METHOD VisitComponent
VAR_INPUT
	Component : Core.I_Component;
END_VAR
_OK := TRUE;
IF __QUERYINTERFACE(Component, SafetyComponent) THEN
	IF NOT SafetyComponent.OK THEN
		ErrorComponent := Component;
		_OK			   := FALSE;
	END_IF
END_IF
END_METHOD

END_FUNCTION_BLOCK

// Components/Safety/Visitor/SetSafetySimulationVisitor
FUNCTION_BLOCK SetSafetySimulationVisitor IMPLEMENTS I_ComponentVisitor
VAR
	SafetyComponent : I_SafetyBase;
	InfoData		: ST_SafetyStateDiag;
	_Simulated		: BOOL;
END_VAR

PROPERTY Diag : UINT
SET
InfoData.Diag := Diag;
END_SET
END_PROPERTY

PROPERTY Simulated : BOOL
GET
Simulated := _Simulated;
END_GET
SET
_Simulated := Simulated;
END_SET
END_PROPERTY

PROPERTY State : USINT
SET
InfoData.State := State;
END_SET
END_PROPERTY

METHOD VisitComponent
VAR_INPUT
	Component : Core.I_Component;
END_VAR
IF __QUERYINTERFACE(Component, SafetyComponent) THEN
	SafetyComponent.Simulated := _Simulated;
	SafetyComponent.SimulateSafetyDiag(InfoData.Diag);
	SafetyComponent.SimulateSafetyState(InfoData.State);
END_IF
END_METHOD

END_FUNCTION_BLOCK

// Components/Safety/SafetyAndOrFB
FUNCTION_BLOCK SafetyAndOrFB EXTENDS SafetyBase
VAR
END_VAR

METHOD CyclicLogic
VAR_INST
	LinkError : BOOL;
END_VAR
SUPER^.CyclicLogic();
_OK := SUPER^.InfoData.State = E_SafetyOrAnd_State.Run;
END_METHOD

END_FUNCTION_BLOCK

// Components/Safety/SafetyBase
FUNCTION_BLOCK SafetyBase EXTENDS CyclicComponent IMPLEMENTS I_SafetyBase
VAR
	InfoData AT %I* : ST_SafetyStateDiag;
	{attribute 'hide'}
	_Simulated : BOOL;
	{attribute 'hide'}
	_OK : BOOL;
	{attribute 'hide'}
	_Error : BOOL;
	{attribute 'hide'}
	_Busy : BOOL;
	{attribute 'hide'}
	_ErrorId	   : UDINT;
	_ResetFunction : I_SafetyReset;
END_VAR

METHOD CyclicLogic
VAR_INST
	LinkError : BOOL;
END_VAR
IF NOT LinkError AND NOT Simulated AND (F_GetMappingStatus(ADR(InfoData), SIZEOF(InfoData)) = EplcMappingStatus.MS_Unmapped) THEN
	LinkError := TRUE;
	Trace.LogMessage(Name, 'Not mapped to Safety, no diagnostics available!');
END_IF

IF _ResetFunction <> 0 THEN
	_ResetFunction.CyclicLogic();
END_IF
END_METHOD

{attribute 'monitoring' := 'call'}
PROPERTY OK : BOOL
GET
OK := _OK;
END_GET
END_PROPERTY

METHOD Reset
IF _ResetFunction <> 0 THEN
	_ResetFunction.Execute();
END_IF
END_METHOD

PROPERTY ResetFunction : I_SafetyReset
SET
_ResetFunction := ResetFunction;
END_SET
END_PROPERTY

{attribute 'monitoring' := 'call'}
PROPERTY Simulated : BOOL
GET
Simulated := _Simulated;
END_GET
SET
_Simulated := Simulated;
END_SET
END_PROPERTY

METHOD SimulateSafetyDiag
VAR_INPUT
	SimulationValueDiag : UINT;
END_VAR
Infodata.Diag := SimulationValueDiag;
END_METHOD

METHOD SimulateSafetyState
VAR_INPUT
	SimulationValueState : USINT;
END_VAR
Infodata.State := SimulationValueState;
END_METHOD

{attribute 'monitoring' := 'call'}
PROPERTY Busy : BOOL
GET
Busy := _Busy;
END_GET
END_PROPERTY

{attribute 'monitoring' := 'call'}
PROPERTY Error : BOOL
GET
Error := _Error;
END_GET
END_PROPERTY

{attribute 'monitoring' := 'call'}
PROPERTY ErrorId : UDINT
GET
ErrorId := _ErrorId;
END_GET
END_PROPERTY

END_FUNCTION_BLOCK

// Components/Safety/SafetyConnectionFB_TcEvents
FUNCTION_BLOCK SafetyConnectionFB_TcEvents EXTENDS SafetyBase IMPLEMENTS I_EventReactionTcEvents
VAR
	Events : TcEventClass('FSoE Connection Events');
END_VAR

METHOD CyclicLogic
VAR_INST
	DiagWord	: WORD;
	BitMaskDiag : WORD := 16#000F;
END_VAR
SUPER^.CyclicLogic();
_OK	   := SUPER^.InfoData.State = E_SafetyConnection_State.Data;
_Error := GetHighestActiveEventReaction() >= TcEventSeverity.Error;
IF _ResetFunction <> 0 AND_THEN _ResetFunction.Busy THEN
	RETURN;
END_IF

BitMaskDiag := 16#000F;
DiagWord	:= TO_WORD(SUPER^.InfoData.Diag) AND BitMaskDiag;
IF (DiagWord = 1) THEN
	Events.RaiseEvent(E_SafetyConnection.InvalidCommand);
END_IF

IF (DiagWord = 2) THEN
	Events.RaiseEvent(E_SafetyConnection.UnknownCommand);
END_IF

IF (DiagWord = 3) THEN
	Events.RaiseEvent(E_SafetyConnection.InvalidConID);
END_IF

IF (DiagWord = 4) THEN
	Events.RaiseEvent(E_SafetyConnection.InvalidCrc);
END_IF

IF (DiagWord = 5) THEN
	Events.RaiseEvent(E_SafetyConnection.WatchdogExpired);
END_IF

IF (DiagWord = 6) THEN
	Events.RaiseEvent(E_SafetyConnection.InvalidFSOEAddr);
END_IF

IF (DiagWord = 7) THEN
	Events.RaiseEvent(E_SafetyConnection.InvalidData);
END_IF

IF (DiagWord = 8) THEN
	Events.RaiseEvent(E_SafetyConnection.InvalidComParameterLen);
END_IF

IF (DiagWord = 9) THEN
	Events.RaiseEvent(E_SafetyConnection.InavlidComParameter);
END_IF

IF (DiagWord = 10) THEN
	Events.RaiseEvent(E_SafetyConnection.InvalidUserParameterLen);
END_IF

IF (DiagWord = 11) THEN
	Events.RaiseEvent(E_SafetyConnection.InvalidUserParameter);
END_IF

IF (DiagWord = 12) THEN
	Events.RaiseEvent(E_SafetyConnection.FSoEMasterReset);
END_IF

IF (DiagWord = 13) THEN
	Events.RaiseEvent(E_SafetyConnection.ModuleErrorOnSlave);
END_IF

IF (DiagWord = 14) THEN
	Events.RaiseEvent(E_SafetyConnection.ModuleError);
END_IF

IF (DiagWord = 15) THEN
	Events.RaiseEvent(E_SafetyConnection.SlaveNotStarted);
END_IF

BitMaskDiag := 16#0010;
DiagWord	:= TO_WORD(SUPER^.InfoData.Diag) AND BitMaskDiag;
IF DiagWord.4 THEN
	Events.RaiseEvent(E_SafetyConnection.FsoESlaveError);
END_IF

BitMaskDiag := 16#0020;
DiagWord	:= TO_WORD(SUPER^.InfoData.Diag) AND BitMaskDiag;
IF DiagWord.5 THEN
	Events.RaiseEvent(E_SafetyConnection.FsoESlaveFailSafeValue);
END_IF

BitMaskDiag := 16#0040;
DiagWord	:= TO_WORD(SUPER^.InfoData.Diag) AND BitMaskDiag;
IF DiagWord.6 THEN
	Events.RaiseEvent(E_SafetyConnection.Startup);
END_IF

BitMaskDiag := 16#0080;
DiagWord	:= TO_WORD(SUPER^.InfoData.Diag) AND BitMaskDiag;
IF DiagWord.7 THEN
	Events.RaiseEvent(E_SafetyConnection.FsoEMasterSafeValue);
END_IF

IF SUPER^.InfoData.Diag.3 THEN
	Events.RaiseEvent(E_SafetyEstop.Disc4);
END_IF

IF SUPER^.InfoData.Diag.4 THEN
	Events.RaiseEvent(E_SafetyEstop.EDM1);
END_IF

IF SUPER^.InfoData.Diag.5 THEN
	Events.RaiseEvent(E_SafetyEstop.EDM2);
END_IF
END_METHOD

METHOD GetHighestActiveEventReaction : DINT
GetHighestActiveEventReaction := Events.GetHighestActiveEventReaction();
END_METHOD

METHOD GetHighestActiveEventSeverity : Core.TcEventSeverity
GetHighestActiveEventSeverity := Events.GetHighestActiveEventSeverity();
END_METHOD

METHOD Reset
SUPER^.Reset();
Events.Reset();
END_METHOD

METHOD SetEventReactions
VAR_INPUT
	Verbose	 : DINT := 0;
	Info	 : DINT := 1;
	Warning	 : DINT := 2;
	Error	 : DINT := 3;
	Critical : DINT := 4;
END_VAR
Events.SetEventReactions(Verbose,
						 Info,
						 Warning,
						 Error,
						 Critical);
END_METHOD

(*FB_Init is always available implicitly and it is used primarily for initialization.
The return value is not evaluated. For a specific influence, you can also declare the
methods explicitly and provide additional code there with the standard initialization
code. You can evaluate the return value.*)
METHOD FB_Init : BOOL
VAR_INPUT
	(* TRUE: the retain variables are initialized (reset warm / reset cold)*)
	bInitRetains : BOOL;

	(* TRUE: the instance will be copied to the copy code afterward (online change)   *)
	bInCopyCode : BOOL;
	Name		: Core.T_MaxString;
END_VAR
Events.GenerateTcEvents(Name, ADR(TC_events.SafetyConnection), SIZEOF(ST_SafetyConnection));
END_METHOD

END_FUNCTION_BLOCK

// Components/Safety/SafetyEdmFB_TcEvents
FUNCTION_BLOCK SafetyEdmFB_TcEvents EXTENDS SafetyBase IMPLEMENTS I_EventReactionTcEvents, I_InSafetyGroup
VAR
	Events		 : TcEventClass('Safety EDM Events');
	_SafetyGroup : I_TaskResult;
END_VAR

METHOD CyclicLogic
SUPER^.CyclicLogic();
_OK	   := SUPER^.InfoData.State <> E_SafetyEdm_State.Error;
_Error := GetHighestActiveEventReaction() >= TcEventSeverity.Error;
IF _SafetyGroup <> 0 THEN
	IF _SafetyGroup.Error THEN
		Events.Reset();
		RETURN;
	END_IF
END_IF

IF _ResetFunction <> 0 AND_THEN _ResetFunction.Busy THEN
	RETURN;
END_IF

IF SUPER^.InfoData.Diag.0 THEN
	Events.RaiseEvent(E_SafetyEdm.SwitchOffTime);
END_IF

IF SUPER^.InfoData.Diag.1 THEN
	Events.RaiseEvent(E_SafetyEdm.SwitchOnTime);
END_IF
END_METHOD

METHOD GetHighestActiveEventReaction : DINT
GetHighestActiveEventReaction := Events.GetHighestActiveEventReaction();
END_METHOD

METHOD GetHighestActiveEventSeverity : Core.TcEventSeverity
GetHighestActiveEventSeverity := Events.GetHighestActiveEventSeverity();
END_METHOD

METHOD Reset
SUPER^.Reset();
Events.Reset();
END_METHOD

METHOD SetEventReactions
VAR_INPUT
	Verbose	 : DINT := 0;
	Info	 : DINT := 1;
	Warning	 : DINT := 2;
	Error	 : DINT := 3;
	Critical : DINT := 4;
END_VAR
Events.SetEventReactions(Verbose,
						 Info,
						 Warning,
						 Error,
						 Critical);
END_METHOD

(*FB_Init is always available implicitly and it is used primarily for initialization.
The return value is not evaluated. For a specific influence, you can also declare the
methods explicitly and provide additional code there with the standard initialization
code. You can evaluate the return value.*)
METHOD FB_Init : BOOL
VAR_INPUT
	(* TRUE: the retain variables are initialized (reset warm / reset cold)*)
	bInitRetains : BOOL;

	(* TRUE: the instance will be copied to the copy code afterward (online change)   *)
	bInCopyCode : BOOL;
	Name		: Core.T_MaxString;
END_VAR
Events.GenerateTcEvents(Name, ADR(TC_events.SafetyEdm), SIZEOF(ST_SafetyEdm));
END_METHOD

PROPERTY SafetyGroup : I_TaskResult
SET
_SafetyGroup := SafetyGroup;
END_SET
END_PROPERTY

END_FUNCTION_BLOCK

// Components/Safety/SafetyEstopFB_TcEvents
FUNCTION_BLOCK SafetyEstopFB_TcEvents EXTENDS SafetyBase IMPLEMENTS I_EventReactionTcEvents, I_InSafetyGroup
VAR
	{attribute 'hide'}
	_ActiveName	 : STRING := 'pressed!';
	Events		 : TcEventClass('Safety E-Stop Events');
	_SafetyGroup : I_TaskResult;
END_VAR

METHOD CyclicLogic
SUPER^.CyclicLogic();
_OK	   := SUPER^.InfoData.State = E_SafetyEStop_State.Run;
_Error := GetHighestActiveEventReaction() >= TcEventSeverity.Error;
IF _SafetyGroup <> 0 THEN
	IF _SafetyGroup.Error THEN
		Events.Reset();
		RETURN;
	END_IF
END_IF

IF _ResetFunction <> 0 AND_THEN _ResetFunction.Busy THEN
	RETURN;
END_IF

IF NOT SUPER^.OK THEN
	Events.Arguments(E_SafetyEstop.Active).Clear().AddString(_ActiveName);
	Events.RaiseEvent(E_SafetyEstop.Active);
END_IF

IF SUPER^.InfoData.Diag.0 THEN
	Events.RaiseEvent(E_SafetyEstop.Disc1);
END_IF

IF SUPER^.InfoData.Diag.1 THEN
	Events.RaiseEvent(E_SafetyEstop.Disc2);
END_IF

IF SUPER^.InfoData.Diag.2 THEN
	Events.RaiseEvent(E_SafetyEstop.Disc3);
END_IF

IF SUPER^.InfoData.Diag.3 THEN
	Events.RaiseEvent(E_SafetyEstop.Disc4);
END_IF

IF SUPER^.InfoData.Diag.4 THEN
	Events.RaiseEvent(E_SafetyEstop.EDM1);
END_IF

IF SUPER^.InfoData.Diag.5 THEN
	Events.RaiseEvent(E_SafetyEstop.EDM2);
END_IF
END_METHOD

METHOD GetHighestActiveEventReaction : DINT
GetHighestActiveEventReaction := Events.GetHighestActiveEventReaction();
END_METHOD

METHOD GetHighestActiveEventSeverity : Core.TcEventSeverity
GetHighestActiveEventSeverity := Events.GetHighestActiveEventSeverity();
END_METHOD

METHOD Reset
SUPER^.Reset();
Events.Reset();
END_METHOD

METHOD SetEventReactions
VAR_INPUT
	Verbose	 : DINT := 0;
	Info	 : DINT := 1;
	Warning	 : DINT := 2;
	Error	 : DINT := 3;
	Critical : DINT := 4;
END_VAR
Events.SetEventReactions(Verbose,
						 Info,
						 Warning,
						 Error,
						 Critical);
END_METHOD

{attribute 'monitoring' := 'call'}
PROPERTY ActiveName : STRING
SET
_ActiveName := ActiveName;
END_SET
END_PROPERTY

(*FB_Init is always available implicitly and it is used primarily for initialization.
The return value is not evaluated. For a specific influence, you can also declare the
methods explicitly and provide additional code there with the standard initialization
code. You can evaluate the return value.*)
METHOD FB_Init : BOOL
VAR_INPUT
	(* TRUE: the retain variables are initialized (reset warm / reset cold)*)
	bInitRetains : BOOL;

	(* TRUE: the instance will be copied to the copy code afterward (online change)   *)
	bInCopyCode : BOOL;
	Name		: Core.T_MaxString;
END_VAR
Events.GenerateTcEvents(Name, ADR(TC_events.SafetyEstop), SIZEOF(ST_SafetyEstop));
END_METHOD

PROPERTY SafetyGroup : I_TaskResult
SET
_SafetyGroup := SafetyGroup;
END_SET
END_PROPERTY

END_FUNCTION_BLOCK

// Components/Safety/SafetyGroup_TcEvents
FUNCTION_BLOCK SafetyGroup_TcEvents EXTENDS SafetyBase IMPLEMENTS I_EventReactionTcEvents
VAR
	Run AT %Q* : BOOL;
	Events	   : TcEventClass('Safety Group Events');
	{attribute 'hide'}
	_AutoResetFaults : BOOL;
END_VAR

METHOD CyclicLogic
VAR_INST
	LinkErrorRun	 : BOOL;
	AutoFaultAck	 : TON;
	TriggerAutoReset : R_TRIG;
END_VAR
SUPER^.CyclicLogic();
IF NOT LinkErrorRun AND NOT Simulated AND (F_GetMappingStatus(ADR(Run), SIZEOF(Run)) = EplcMappingStatus.MS_Unmapped) THEN
	LinkErrorRun := TRUE;
	Trace.LogMessage(Name, 'Group Run not mapped to Safety!');
END_IF

Run := TRUE;
IF _ResetFunction <> 0 THEN
	AutoFaultAck(IN := (_AutoResetFaults AND (SUPER^.InfoData.Diag <> 0)) AND NOT _ResetFunction.Busy, PT := T#250MS);
	TriggerAutoReset(CLK := AutoFaultAck.Q);
	IF TriggerAutoReset.Q THEN
		_ResetFunction.Execute();
	END_IF

	_Busy := _ResetFunction.Busy;
END_IF

_OK	   := SUPER^.InfoData.State = E_SafetyGroup_State.Run;
_Error := GetHighestActiveEventReaction() >= TcEventSeverity.Error;
IF _ResetFunction <> 0 AND_THEN _ResetFunction.Busy THEN
	RETURN;
END_IF

IF SUPER^.InfoData.Diag = E_SafetyGroup_Diag.FbError THEN
	Events.RaiseEvent(E_SafetyGroup.FbError);
END_IF

IF SUPER^.InfoData.Diag = E_SafetyGroup_Diag.ComError THEN
	Events.RaiseEvent(E_SafetyGroup.ComError);
END_IF

IF SUPER^.InfoData.Diag = E_SafetyGroup_Diag.ModuleError THEN
	Events.RaiseEvent(E_SafetyGroup.ModuleError);
END_IF

IF SUPER^.InfoData.Diag = E_SafetyGroup_Diag.CmpError THEN
	Events.RaiseEvent(E_SafetyGroup.ModuleError);
END_IF

IF SUPER^.InfoData.Diag = E_SafetyGroup_Diag.DeactiveError THEN
	Events.RaiseEvent(E_SafetyGroup.DeactiveError);
END_IF

IF SUPER^.InfoData.Diag = E_SafetyGroup_Diag.RestartError THEN
	Events.RaiseEvent(E_SafetyGroup.RestartError);
END_IF
END_METHOD

METHOD GetHighestActiveEventReaction : DINT
GetHighestActiveEventReaction := Events.GetHighestActiveEventReaction();
END_METHOD

METHOD GetHighestActiveEventSeverity : Core.TcEventSeverity
GetHighestActiveEventSeverity := Events.GetHighestActiveEventSeverity();
END_METHOD

METHOD Reset
SUPER^.Reset();
Events.Reset();
END_METHOD

METHOD SetEventReactions
VAR_INPUT
	Verbose	 : DINT := 0;
	Info	 : DINT := 1;
	Warning	 : DINT := 2;
	Error	 : DINT := 3;
	Critical : DINT := 4;
END_VAR
Events.SetEventReactions(Verbose,
						 Info,
						 Warning,
						 Error,
						 Critical);
END_METHOD

{attribute 'monitoring' := 'call'}
PROPERTY AutoResetFaults : BOOL
GET
AutoResetFaults := _AutoResetFaults;
END_GET
SET
_AutoResetFaults := AutoResetFaults;
END_SET
END_PROPERTY

(*FB_Init is always available implicitly and it is used primarily for initialization.
The return value is not evaluated. For a specific influence, you can also declare the
methods explicitly and provide additional code there with the standard initialization
code. You can evaluate the return value.*)
METHOD FB_Init : BOOL
VAR_INPUT
	(* TRUE: the retain variables are initialized (reset warm / reset cold)*)
	bInitRetains : BOOL;

	(* TRUE: the instance will be copied to the copy code afterward (online change)   *)
	bInCopyCode : BOOL;
	Name		: Core.T_MaxString;
END_VAR
Events.GenerateTcEvents(Name, ADR(TC_events.SafetyGroup), SIZEOF(ST_SafetyGroup));
END_METHOD

END_FUNCTION_BLOCK

// Components/Safety/SafetyModule
FUNCTION_BLOCK SafetyModule EXTENDS Module IMPLEMENTS I_SafetyModule
VAR
	SequenceState			 : UDINT;
	TwinSAFEResetDelay		 : TON;
	SafetyPLC_WcState AT %I* : BOOL;
	SafetyPLC_AmsAddr AT %I* : AMSADDR;
	_SafetyPlcCoE			 : CoeDevice('Safety PLC') := (AdsAddr := SafetyPLC_AmsAddr);
	_SafetyAddressInfo		 : ST_SafetyAddressInfo;
END_VAR

VAR
	GetComponentsTaskResultVisitor : GetComponentsTaskResultVisitor;
	SetSafetySimulationVisitor	   : SetSafetySimulationVisitor;
	SafetyOkVisitor				   : SafetyOkVisitor;
END_VAR

METHOD OnCyclicCall
IF NOT Initialized THEN
	Initialize();
	RETURN;
END_IF

TwinSAFEResetDelay(PT := T#250MS);
CASE SequenceState OF
	0:
		TwinSAFEResetDelay.IN := FALSE;

	10:
		ResetComponents();
		SequenceState := 20;

	20:
		TwinSAFEResetDelay.IN := TRUE;
		IF TwinSAFEResetDelay.Q THEN
			SequenceState := 0;
		END_IF
END_CASE

GetComponentsTaskResultVisitor.Update(THIS^);
THIS^.Components.Accept(SafetyOkVisitor);
END_METHOD

(* This Module will be done initialize when ModuleInitialized := TRUE;, subequently all subitems will be called to be initialized *)
METHOD Initializing
_SafetyPlcCoE.CyclicLogic();
CASE SequenceState OF
	0:
		IF F_GetMappingStatus(ADR(SafetyPLC_WcState), SIZEOF(SafetyPLC_WcState)) = EplcMappingStatus.MS_Unmapped OR F_GetMappingStatus(ADR(SafetyPLC_AmsAddr), SIZEOF(SafetyPLC_AmsAddr)) = EplcMappingStatus.MS_Unmapped THEN
			SequenceState := 100;
			Trace.LogMessage(Name, 'Safety PLC not mapped, info will not be read!');
		ELSE
			SequenceState := SequenceState + 10;
		END_IF

	10:
		IF NOT SafetyPLC_WcState THEN
			SequenceState := SequenceState + 10;
		END_IF

	20:
		SafetyPlcCoE.Read(16#F980,
						  1,
						  ADR(_SafetyAddressInfo.FSoEAddress),
						  SIZEOF(_SafetyAddressInfo.FSoEAddress));

		SequenceState := SequenceState + 1;

	21:
		IF NOT SafetyPlcCoE.Error AND NOT SafetyPlcCoE.Busy THEN
			SequenceState := SequenceState + 1;
		END_IF

	22:
		SafetyPlcCoE.Read(16#F980,
						  2,
						  ADR(_SafetyAddressInfo.SerialNumber),
						  SIZEOF(_SafetyAddressInfo.SerialNumber));

		SequenceState := SequenceState + 1;

	23:
		IF NOT SafetyPlcCoE.Error AND NOT SafetyPlcCoE.Busy THEN
			SequenceState := SequenceState + 1;
		END_IF

	24:
		SafetyPlcCoE.Read(16#F980,
						  3,
						  ADR(_SafetyAddressInfo.ProjectCRC),
						  SIZEOF(_SafetyAddressInfo.ProjectCRC));

		SequenceState := SequenceState + 1;

	25:
		IF NOT SafetyPlcCoE.Error AND NOT SafetyPlcCoE.Busy THEN
			SequenceState := SequenceState + 1;
		END_IF

	26:
		SafetyPlcCoE.Read(16#F980,
						  4,
						  ADR(_SafetyAddressInfo.DefaultProjectCRC),
						  SIZEOF(_SafetyAddressInfo.DefaultProjectCRC));

		SequenceState := SequenceState + 1;

	27:
		IF NOT SafetyPlcCoE.Error AND NOT SafetyPlcCoE.Busy THEN
			SequenceState := 100;
		END_IF

	100:
		SequenceState	  := 0;
		ModuleInitialized := TRUE;
END_CASE
END_METHOD

{attribute 'monitoring' := 'call'}
PROPERTY Simulated : BOOL
GET
Simulated := SetSafetySimulationVisitor.Simulated;
END_GET
SET
SetSafetySimulationVisitor.Simulated := Simulated;
Components.Accept(SetSafetySimulationVisitor);
END_SET
END_PROPERTY

METHOD SimulateSafetyDiag
VAR_INPUT
	SimulationValueDiag : UINT;
END_VAR
SetSafetySimulationVisitor.Diag := SimulationValueDiag;
Components.Accept(SetSafetySimulationVisitor);
END_METHOD

METHOD SimulateSafetyState
VAR_INPUT
	SimulationValueState : USINT;
END_VAR
SetSafetySimulationVisitor.State := SimulationValueState;
Components.Accept(SetSafetySimulationVisitor);
END_METHOD

{attribute 'monitoring' := 'call'}
PROPERTY Busy : BOOL
GET
Busy := SequenceState <> 0;
END_GET
END_PROPERTY

{attribute 'monitoring' := 'call'}
PROPERTY Error : BOOL
GET
Error := GetComponentsTaskResultVisitor.Error;
END_GET
END_PROPERTY

{attribute 'monitoring' := 'call'}
PROPERTY ErrorId : UDINT
GET
ErrorId := GetComponentsTaskResultVisitor.ErrorId;
END_GET
END_PROPERTY

METHOD AddSafetyComponent
VAR_INPUT
	Component : I_SafetyBase;
END_VAR
Component.RegisterWithParent(THIS^);
END_METHOD

(*FB_Init is always available implicitly and it is used primarily for initialization.
The return value is not evaluated. For a specific influence, you can also declare the
methods explicitly and provide additional code there with the standard initialization
code. You can evaluate the return value.*)
METHOD FB_Init : BOOL
VAR_INPUT
	(* TRUE: the retain variables are initialized (reset warm / reset cold)*)
	bInitRetains : BOOL;

	(* TRUE: the instance will be copied to the copy code afterward (online change)   *)
	bInCopyCode : BOOL;
	Name		: Core.T_MaxString;
END_VAR
SafetyPlcCoE.RegisterWithParent(THIS^);
END_METHOD

{attribute 'monitoring' := 'call'}
PROPERTY OK : BOOL
GET
OK := SafetyOkVisitor.OK;
END_GET
END_PROPERTY

METHOD Reset
IF Busy THEN
	RETURN;
END_IF

SequenceState := 10;
END_METHOD

PROPERTY SafetyAddressInfo : REFERENCE TO ST_SafetyAddressInfo
GET
SafetyAddressInfo REF= _SafetyAddressInfo;
END_GET
END_PROPERTY

PROPERTY SafetyPlcCoE : I_CoeDevice
GET
SafetyPlcCoE := _SafetyPlcCoE;
END_GET
END_PROPERTY

END_FUNCTION_BLOCK

// Components/Safety/SafetyMonFB_TcEvents
FUNCTION_BLOCK SafetyMonFB_TcEvents EXTENDS SafetyBase IMPLEMENTS I_EventReactionTcEvents, I_InSafetyGroup
VAR
	{attribute 'hide'}
	_ActiveAlarm : BOOL := TRUE;
	{attribute 'hide'}
	_ActiveName	 : STRING := 'pressed!';
	Events		 : TcEventClass('Safety MonFB Events');
	_SafetyGroup : I_TaskResult;
END_VAR

METHOD CyclicLogic
SUPER^.CyclicLogic();
_OK	   := SUPER^.InfoData.State = E_SafetyEStop_State.Run;
_Error := GetHighestActiveEventReaction() >= TcEventSeverity.Error;
IF _SafetyGroup <> 0 THEN
	IF _SafetyGroup.Error THEN
		Events.Reset();
		RETURN;
	END_IF
END_IF

IF _ResetFunction <> 0 AND_THEN _ResetFunction.Busy THEN
	RETURN;
END_IF

IF NOT SUPER^.OK AND _ActiveAlarm THEN
	Events.Arguments(E_SafetyMon.Active).Clear().AddString(_ActiveName);
	Events.RaiseEvent(E_SafetyMon.Active);
END_IF

IF SUPER^.InfoData.Diag.0 THEN
	Events.RaiseEvent(E_SafetyMon.Disc1);
END_IF

IF SUPER^.InfoData.Diag.1 THEN
	Events.RaiseEvent(E_SafetyMon.Disc2);
END_IF

IF SUPER^.InfoData.Diag.3 THEN
	Events.RaiseEvent(E_SafetyMon.DiscInput);
END_IF

IF SUPER^.InfoData.Diag.4 THEN
	Events.RaiseEvent(E_SafetyMon.Edm1);
END_IF

IF SUPER^.InfoData.Diag.5 THEN
	Events.RaiseEvent(E_SafetyMon.Edm2);
END_IF

IF SUPER^.InfoData.Diag.8 THEN
	Events.RaiseEvent(E_SafetyMon.Disc1Safe);
END_IF

IF SUPER^.InfoData.Diag.9 THEN
	Events.RaiseEvent(E_SafetyMon.Disc2Safe);
END_IF

IF SUPER^.InfoData.Diag.10 THEN
	Events.RaiseEvent(E_SafetyMon.DiscInputSafe);
END_IF
END_METHOD

METHOD GetHighestActiveEventReaction : DINT
GetHighestActiveEventReaction := Events.GetHighestActiveEventReaction();
END_METHOD

METHOD GetHighestActiveEventSeverity : Core.TcEventSeverity
GetHighestActiveEventSeverity := Events.GetHighestActiveEventSeverity();
END_METHOD

METHOD Reset
SUPER^.Reset();
Events.Reset();
END_METHOD

METHOD SetEventReactions
VAR_INPUT
	Verbose	 : DINT := 0;
	Info	 : DINT := 1;
	Warning	 : DINT := 2;
	Error	 : DINT := 3;
	Critical : DINT := 4;
END_VAR
Events.SetEventReactions(Verbose,
						 Info,
						 Warning,
						 Error,
						 Critical);
END_METHOD

PROPERTY ActiveAlarm : BOOL
SET
_ActiveAlarm := ActiveAlarm;
END_SET
END_PROPERTY

PROPERTY ActiveName : STRING
SET
_ActiveName := ActiveName;
END_SET
END_PROPERTY

(*FB_Init is always available implicitly and it is used primarily for initialization.
The return value is not evaluated. For a specific influence, you can also declare the
methods explicitly and provide additional code there with the standard initialization
code. You can evaluate the return value.*)
METHOD FB_Init : BOOL
VAR_INPUT
	(* TRUE: the retain variables are initialized (reset warm / reset cold)*)
	bInitRetains : BOOL;

	(* TRUE: the instance will be copied to the copy code afterward (online change)   *)
	bInCopyCode : BOOL;
	Name		: Core.T_MaxString;
END_VAR
Events.GenerateTcEvents(Name, ADR(TC_events.SafetyMon), SIZEOF(ST_SafetyMon));
END_METHOD

PROPERTY SafetyGroup : I_TaskResult
SET
_SafetyGroup := SafetyGroup;
END_SET
END_PROPERTY

END_FUNCTION_BLOCK

// Components/Tcp Ip/Interface/I_TcpIpConnection
INTERFACE I_TcpIpConnection EXTENDS I_Component

{attribute 'monitoring' := 'call'}
PROPERTY IP : T_IPv4Addr
SET
END_SET
END_PROPERTY

{attribute 'monitoring' := 'call'}
PROPERTY Port : UDINT
SET
END_SET
END_PROPERTY

METHOD RegisterCommand
VAR_INPUT
	Command : I_TcpIpSubscription;
END_VAR
END_METHOD

METHOD SendCommand
VAR_INPUT
	Command : STRING(4096);
END_VAR
END_METHOD

METHOD SendPriorityCommand
VAR_INPUT
	Command : STRING(4096);
END_VAR
END_METHOD

END_INTERFACE

// Components/Tcp Ip/Interface/I_TcpIpSubscription
INTERFACE I_TcpIpSubscription EXTENDS I_Base

METHOD UpdateCommandResult
VAR_INPUT
	Response : STRING(4096);
END_VAR
END_METHOD

END_INTERFACE

// Components/Tcp Ip/TcpIpCommand
FUNCTION_BLOCK ABSTRACT TcpIpCommand EXTENDS CyclicComponent IMPLEMENTS I_TcpIpSubscription
VAR
	TcpIpConnection : I_TcpIpConnection;
	{attribute 'hide'}
	_Initialized   : BOOL := FALSE;
	CommandActive  : BOOL;
	CommandTimeout : TON;

	//
	Response	  : STRING(4096);
	Command		  : STRING(4096);
	JsonSaxWriter : FB_JsonSaxWriter;
	JsonDocument  : SJsonValue;
	JsonValue	  : SJsonValue;
	JsonDomParser : FB_JsonDomParser;
END_VAR

METHOD CyclicLogic
CommandTimeout(IN := CommandActive, PT := T#10S);
IF CommandTimeout.Q THEN
	CommandActive := FALSE;
	ADSLOGSTR(ADSLOG_MSGTYPE_HINT, CONCAT('Command response not recieved! ', Name), '');
END_IF
END_METHOD

(*FB_Init is always available implicitly and it is used primarily for initialization.
The return value is not evaluated. For a specific influence, you can also declare the
methods explicitly and provide additional code there with the standard initialization
code. You can evaluate the return value.*)
METHOD FB_Init : BOOL
VAR_INPUT
	(* TRUE: the retain variables are initialized (reset warm / reset cold)*)
	bInitRetains : BOOL;

	(* TRUE: the instance will be copied to the copy code afterward (online change)   *)
	bInCopyCode		: BOOL;
	Name			: Core.T_MaxString;
	TcpIpConnection : I_TcpIpConnection;
END_VAR
THIS^.TcpIpConnection := TcpIpConnection;
TcpIpConnection.RegisterCommand(THIS^);
END_METHOD

METHOD ABSTRACT UpdateCommandResult
VAR_INPUT
	Response : STRING(4096);
END_VAR
END_METHOD

END_FUNCTION_BLOCK

// Components/Tcp Ip/TcpIpConnection
FUNCTION_BLOCK TcpIpConnection EXTENDS CyclicComponent IMPLEMENTS I_TcpIpConnection, I_Initializable
VAR
	_Initialized   : BOOL;
	_IP			   : T_IPv4Addr := '127.0.0.1';
	_Port		   : UDINT;
	SocketCloseAll : FB_SocketCloseAll;

	// Send Port
	ReconnectTimer		   : TON;
	ClientServerConnection : FB_ClientServerConnection;
	ServerConnectionState  : E_SocketConnectionState;
	SocketSend			   : FB_SocketSend;
	SendMessage			   : STRING(4096);
	Socket				   : T_HSOCKET;
	SendDelay			   : TON := (PT := T#100MS);
	PollTimer			   : TON;
	ResponseTimer		   : TON;
	SocketReceive		   : FB_SocketReceive;
	ReceiveMessage		   : STRING(4096);
END_VAR

VAR
	ApiCommands		   : ARRAY[0..COMMAND_BUFFER] OF I_TcpIpSubscription;
	SendBuffer		   : ARRAY[0..COMMAND_BUFFER] OF STRING(4096);
	PrioritySendBuffer : ARRAY[0..COMMAND_BUFFER] OF STRING(4096);
END_VAR

VAR CONSTANT
	RECON_TIME	   : TIME := T#10S;
	COMMAND_BUFFER : DINT := 99;
END_VAR

METHOD CyclicLogic
IF NOT _Initialized THEN
	Initialize();
	RETURN;
END_IF

SendReceiveSequence();
END_METHOD

METHOD Initialize
SocketCloseAll(sSrvNetId := '', bExecute := TRUE);
IF NOT SocketCloseAll.bBusy AND NOT SocketCloseAll.bError THEN
	_Initialized := TRUE;
END_IF
END_METHOD

{attribute 'monitoring' := 'call'}
PROPERTY Initialized : BOOL
GET
Initialized := _Initialized;
END_GET
SET
_Initialized := Initialized;
END_SET
END_PROPERTY

METHOD PROTECTED EvaluateResponse
VAR
	i : DINT;
END_VAR
FOR i := 0 TO COMMAND_BUFFER DO
	IF ApiCommands[i] = 0 THEN
		EXIT;
	END_IF

	ApiCommands[i].UpdateCommandResult(ReceiveMessage);
END_FOR

MEMSET(ADR(ReceiveMessage), 0, SIZEOF(ReceiveMessage));
END_METHOD

METHOD PROTECTED GetNextCommand
VAR
	i : DINT;
END_VAR
IF SendBuffer[0] <> '' THEN
	SendMessage := SendBuffer[0];
	FOR i := 0 TO (COMMAND_BUFFER - 1) DO
		SendBuffer[i] := SendBuffer[i + 1];
	END_FOR
END_IF
END_METHOD

METHOD PROTECTED GetNextPriorityCommand
VAR
	i : DINT;
END_VAR
IF PrioritySendBuffer[0] <> '' THEN
	SendMessage := PrioritySendBuffer[0];
	FOR i := 0 TO (COMMAND_BUFFER - 1) DO
		PrioritySendBuffer[i] := PrioritySendBuffer[i + 1];
	END_FOR
END_IF
END_METHOD

METHOD PROTECTED SendReceiveSequence
VAR_INST
	SequenceState : UDINT;
END_VAR
ClientServerConnection(sSrvNetID   := '',
					   sRemoteHost := _IP,
					   nRemotePort := _Port,
					   hSocket	   => Socket,
					   eState	   => ServerConnectionState);

SocketSend(sSrvNetId := '',
		   hSocket	 := Socket,
		   cbLen	 := TO_UDINT(LEN(SendMessage)),
		   pSrc		 := ADR(SendMessage),
		   tTimeout	 := T#5S);

SocketReceive(sSrvNetId := '',
			  hSocket	:= Socket,
			  cbLen		:= SIZEOF(ReceiveMessage),
			  pDest		:= ADR(ReceiveMessage),
			  tTimeout	:= T#5S);

//
ReconnectTimer(PT := RECON_TIME);
PollTimer(PT := T#100MS);
ResponseTimer(PT := T#50S);
CASE SequenceState OF
	0:
		ClientServerConnection.bEnable := TRUE;
		IF ServerConnectionState = eSOCKET_CONNECTED THEN
			SequenceState := SequenceState + 10;
		END_IF

		IF ClientServerConnection.bError THEN
			ADSLOGSTR(ADSLOG_MSGTYPE_HINT, CONCAT('ClientServerConnection.bError: ', TO_STRING(ClientServerConnection.nErrId)), '');
			SequenceState := 200;
		END_IF

	10:
		// SENDING -----------------------------------------------------------------------------------
		SendDelay(IN := NOT SendDelay.Q);
		IF SendMessage = '' THEN
			GetNextPriorityCommand();
		END_IF

		IF SendMessage = '' THEN
			GetNextCommand();
		END_IF

		IF SocketSend.bExecute AND NOT SocketSend.bBusy AND NOT SocketSend.bError THEN
			ADSLOGSTR(ADSLOG_MSGTYPE_HINT, Concat('Client sent: ', SendMessage), '');
			MEMSET(ADR(SendMessage), 0, SIZEOF(SendMessage));
			SocketSend.bExecute := FALSE;
		END_IF

		IF SendMessage <> '' AND NOT SocketSend.bExecute AND SendDelay.Q THEN
			SocketSend.bExecute := TRUE;
		END_IF

		IF SocketSend.bError THEN
			ADSLOGSTR(ADSLOG_MSGTYPE_HINT, CONCAT('SocketSend.bError: ', TO_STRING(SocketSend.nErrId)), '');
			SequenceState := 200;
		END_IF

		// RECEIVING -----------------------------------------------------------------------------------
		PollTimer.IN		   := TRUE;
		SocketReceive.bExecute := TRUE;
		IF PollTimer.Q AND NOT SocketReceive.bError AND NOT SocketReceive.bBusy THEN
			IF SocketReceive.nRecBytes > 0 THEN
				ResponseTimer.IN := FALSE;
				ADSLOGSTR(ADSLOG_MSGTYPE_HINT, Concat('Client recieved: ', ReceiveMessage), '');
				EvaluateResponse();
			END_IF

			SequenceState := 11;
			// Stale connection, disconnected while socket was open
			IF SocketReceive.nRecBytes = 0 THEN
				ResponseTimer.IN := TRUE;
				IF ResponseTimer.Q THEN
					ADSLOGSTR(ADSLOG_MSGTYPE_HINT, 'Receive Connection stale - re-connect!', '');
					SequenceState := 200;
				END_IF
			END_IF
		END_IF

		IF SocketReceive.bError THEN
			ADSLOGSTR(ADSLOG_MSGTYPE_HINT, CONCAT('SocketReceive.bError: ', TO_STRING(SocketReceive.nErrId)), '');
			SequenceState := 200;
		END_IF

	11:
		PollTimer.IN		   := FALSE;
		SocketReceive.bExecute := FALSE;
		SequenceState		   := 10;

	200:
		ReconnectTimer.IN			   := TRUE;
		ResponseTimer.IN			   := FALSE;
		ClientServerConnection.bEnable := FALSE;
		IF ServerConnectionState = eSOCKET_DISCONNECTED AND ReconnectTimer.Q THEN
			ReconnectTimer.IN := FALSE;
			SequenceState	  := 0;
		END_IF
END_CASE
END_METHOD

{attribute 'monitoring' := 'call'}
PROPERTY IP : T_IPv4Addr
SET
_IP := IP;
END_SET
END_PROPERTY

{attribute 'monitoring' := 'call'}
PROPERTY Port : UDINT
SET
_Port := Port;
END_SET
END_PROPERTY

METHOD RegisterCommand
VAR_INPUT
	Command : I_TcpIpSubscription;
END_VAR

VAR
	i : DINT;
END_VAR
FOR i := 0 TO COMMAND_BUFFER DO
	IF ApiCommands[i] = 0 THEN
		ApiCommands[i] := Command;
		RETURN;
	END_IF
END_FOR
END_METHOD

METHOD SendCommand
VAR_INPUT
	Command : STRING(4096);
END_VAR

VAR
	i : DINT;
END_VAR
FOR i := 0 TO COMMAND_BUFFER DO
	IF SendBuffer[i] = '' THEN
		SendBuffer[i] := Command;
		RETURN;
	END_IF
END_FOR
END_METHOD

METHOD SendPriorityCommand
VAR_INPUT
	Command : STRING(4096);
END_VAR

VAR
	i : DINT;
END_VAR
FOR i := 0 TO COMMAND_BUFFER DO
	IF PrioritySendBuffer[i] = '' THEN
		PrioritySendBuffer[i] := Command;
		RETURN;
	END_IF
END_FOR
END_METHOD

END_FUNCTION_BLOCK

// Project Information/F_GetCompany
// This function has been automatically generated from the project information.
{attribute 'signature_flag' := '1073741824'}
{attribute 'TcGenerated'}
{attribute 'no-analysis'}
FUNCTION F_GetCompany : WSTRING
VAR_INPUT
	
END_VAR

F_GetCompany := "Beckhoff Automation LLC";

END_FUNCTION

// Project Information/F_GetTitle
// This function has been automatically generated from the project information.
{attribute 'signature_flag' := '1073741824'}
{attribute 'TcGenerated'}
{attribute 'no-analysis'}
FUNCTION F_GetTitle : WSTRING
VAR_INPUT
	
END_VAR

F_GetTitle := "CoreComponents";

END_FUNCTION

// Project Information/F_GetVersion
// This function has been automatically generated from the project information.
{attribute 'signature_flag' := '1073741824'}
{attribute 'TcGenerated'}
{attribute 'no-analysis'}
FUNCTION F_GetVersion : ST_LibVersion
VAR_INPUT
	
END_VAR

F_GetVersion.iMajor := 1;
F_GetVersion.iMinor := 1;
F_GetVersion.iBuild := 9;
F_GetVersion.iRevision := 0;
F_GetVersion.sVersion := '1.1.9';
F_GetVersion.nFlags := 0;

END_FUNCTION

// Utilities/File/Interface/I_FileHandler
INTERFACE I_FileHandler EXTENDS I_Component, I_Cyclic, I_TaskResult, I_TaskResult, I_Resettable

METHOD ClearDocument
VAR_INPUT
END_VAR
END_METHOD

PROPERTY Datatype : T_MaxString
SET
END_SET
END_PROPERTY

METHOD LoadFile
END_METHOD

PROPERTY nData : UDINT
SET
END_SET
END_PROPERTY

PROPERTY PUBLIC Path : T_MaxString
GET
END_GET
SET
END_SET
END_PROPERTY

PROPERTY pData : PVOID
SET
END_SET
END_PROPERTY

METHOD ReadSymbol
END_METHOD

METHOD SaveFile
END_METHOD

PROPERTY SymbolName : T_MaxString
SET
END_SET
END_PROPERTY

PROPERTY Timeout : TIME
SET
END_SET
END_PROPERTY

METHOD UpdateSymbol
END_METHOD

END_INTERFACE

// Utilities/File/File_HMI
FUNCTION_BLOCK File_HMI EXTENDS HmiFunction
VAR
	File : I_FileHandler;
	{ attribute 'TcHmiSymbol.AddSymbol' }
	{ attribute 'TcHmiSymbol.AddSymbol.UserGroups' := '__SystemAdministrators,Admin' }
	File_HMI : ST_File_HMI;
END_VAR

PROPERTY LoadPermissive : I_Permissive
GET
LoadPermissive := File_HMI.Load.Permissive;
END_GET
END_PROPERTY

PROPERTY SavePermissive : I_Permissive
GET
SavePermissive := File_HMI.Save.Permissive;
END_GET
END_PROPERTY

METHOD CyclicLogic
VAR_INST
	SaveRT		 : R_TRIG;
	LoadRT		 : R_TRIG;
	ReloadActive : BOOL;
END_VAR
IF File = 0 THEN
	RETURN;
END_IF

File_HMI.Name		:= File.Name;
File_HMI.HmiEnabled := Enabled;
// HMI Commands
IF Enabled THEN
	SaveRT(CLK := File_HMI.Save.Active);
	IF SaveRT.Q THEN
		IF File_HMI.Save.Permissive.OK THEN
			File.UpdateSymbol();
		END_IF
	END_IF

	IF ReloadActive AND NOT File.Busy AND NOT File.Error THEN
		File.ReadSymbol();
		ReloadActive := FALSE;
	END_IF

	LoadRT(CLK := File_HMI.Load.Active);
	IF LoadRT.Q THEN
		IF File_HMI.Load.Permissive.OK THEN
			File.LoadFile();
			ReloadActive := TRUE;
		END_IF
	END_IF

	IF File_HMI.NewPath THEN
		File.Path		 := File_HMI.Path;
		File_HMI.NewPath := FALSE;
	END_IF
END_IF
END_METHOD

(*FB_Init is always available implicitly and it is used primarily for initialization.
The return value is not evaluated. For a specific influence, you can also declare the
methods explicitly and provide additional code there with the standard initialization
code. You can evaluate the return value.*)
METHOD FB_Init : BOOL
VAR_INPUT
	(* TRUE: the retain variables are initialized (reset warm / reset cold)*)
	bInitRetains : BOOL;

	(* TRUE: the instance will be copied to the copy code afterward (online change)   *)
	bInCopyCode : BOOL;
	Name		: Core.T_MaxString;
	File		: I_FileHandler;
END_VAR
THIS^.File	:= File;
ControlType := 'File';
LinkObject	:= 'File_HMI';
END_METHOD

END_FUNCTION_BLOCK

// Utilities/File/JsonFile
FUNCTION_BLOCK JsonFile
VAR_GENERIC CONSTANT
	FileSize : UDINT := 10000;
END_VAR
EXTENDS CyclicComponent IMPLEMENTS I_FileHandler
VAR
	{attribute 'hide'}
	_Error : BOOL;
	{attribute 'hide'}
	_ErrorId : UDINT;

	//
	_Path	   : STRING;
	TonTimeout : TON;
	_Timeout   : TIME := T#1S;
	SeqLoad	   : UDINT;
	SeqSave	   : UDINT;

	// Folder Management
	CreateDir	 : FB_CreateDir;
	StringHelper : StringHelper;

	// Symbol
	JsonReadWriteDataType : FB_JsonReadWriteDatatype;
	ValueJson			  : STRING(FileSize);
	hr					  : HRESULT;
	_Datatype			  : T_MaxString;
	_SymbolName			  : T_MaxString;
	_nData				  : UDINT;
	_pData				  : PVOID;

	// Json Management 
	FileRead			  : BOOL;
	FileSave			  : BOOL;
	FileLoadOK			  : BOOL;
	FileSaveOK			  : BOOL;
	JsonFileMachineConfig : FB_JsonDomParser;
	JsonDoc				  : SJsonValue;
	JsonProp			  : SJsonValue;
END_VAR

METHOD CyclicLogic
IF _Path <> '' THEN
	FileLoadOK := JsonFileMachineConfig.LoadDocumentFromFile(sFile := _Path, bExec := FileRead);
	FileSaveOK := JsonFileMachineConfig.SaveDocumentToFile(sFile := _Path, bExec := FileSave);
END_IF

TonTimeout(IN := Busy, PT := _Timeout);
IF TonTimeout.Q THEN
	_Error := TRUE;
END_IF

SaveFileSequence();
LoadFileSequence();
END_METHOD

METHOD ClearDocument
VAR_INPUT
END_VAR
JsonDoc := JsonFileMachineConfig.NewDocument();
END_METHOD

PROPERTY Datatype : T_MaxString
SET
_Datatype := Datatype;
END_SET
END_PROPERTY

METHOD LoadFile
IF _Path = '' THEN
	_Error := TRUE;
	Trace.LogMessage(Name, 'File Path not set!');
	RETURN;
END_IF

IF Busy THEN
	RETURN;
END_IF

FileRead := TRUE;
SeqLoad	 := 10;
END_METHOD

PROPERTY nData : UDINT
SET
_nData := nData;
END_SET
END_PROPERTY

PROPERTY PUBLIC Path : T_MaxString
GET
Path := _Path;
END_GET
SET
//Prevent the path from have a space at the end
_Path := Path;
WHILE RIGHT(_Path, 1) = ' ' DO
	_Path := DELETE(_Path, 1, LEN(_Path));
END_WHILE
END_SET
END_PROPERTY

PROPERTY pData : PVOID
SET
_pData := pData;
END_SET
END_PROPERTY

METHOD ReadSymbol
IF JsonDoc = 0 THEN
	Trace.LogMessage(Name, 'Document File not loaded!');
	RETURN;
END_IF

IF _Datatype = '' THEN
	Trace.LogMessage(Name, 'No Datatype specified!');
	RETURN;
END_IF

IF _nData = 0 THEN
	Trace.LogMessage(Name, 'No nData specified!');
	RETURN;
END_IF

IF _pData = 0 THEN
	Trace.LogMessage(Name, 'No pData specified!');
	RETURN;
END_IF

IF _SymbolName = '' THEN
	Trace.LogMessage(Name, 'No PropertyName specified!');
	RETURN;
END_IF

IF Busy THEN
	RETURN;
END_IF

JsonProp := JsonFileMachineConfig.FindMemberPath(JsonDoc, _SymbolName);
JsonFileMachineConfig.CopyJson(v := JsonProp, pDoc := ValueJson, nDoc := SIZEOF(ValueJson));
IF JsonProp <> 0 THEN
	JsonReadWriteDataType.SetSymbolFromJson(sJson		:= ValueJson,
											sDataType	:= _Datatype,
											nData		:= _nData,
											pData		:= _pData,
											hrErrorCode => hr);
ELSE
	THIS^.UpdateSymbol();
END_IF
END_METHOD

METHOD SaveFile
IF _Path = '' THEN
	_Error := TRUE;
	Trace.LogMessage(Name, 'File Path not set!');
	RETURN;
END_IF

IF Busy THEN
	RETURN;
END_IF

FileSave := TRUE;
SeqSave	 := 10;
END_METHOD

PROPERTY SymbolName : T_MaxString
SET
_SymbolName := SymbolName;
END_SET
END_PROPERTY

PROPERTY Timeout : TIME
SET
_Timeout := Timeout;
END_SET
END_PROPERTY

METHOD UpdateSymbol
IF JsonDoc = 0 THEN
	Trace.LogMessage(Name, 'Document File not loaded!');
	RETURN;
END_IF

IF _Datatype = '' THEN
	Trace.LogMessage(Name, 'No Datatype specified!');
	RETURN;
END_IF

IF _nData = 0 THEN
	Trace.LogMessage(Name, 'No nData specified!');
	RETURN;
END_IF

IF _pData = 0 THEN
	Trace.LogMessage(Name, 'No pData specified!');
	RETURN;
END_IF

IF _SymbolName = '' THEN
	Trace.LogMessage(Name, 'No PropertyName specified!');
	RETURN;
END_IF

IF Busy THEN
	RETURN;
END_IF

// Create Json
JsonReadWriteDataType.CopyJsonStringFromSymbol(sDatatype   := _Datatype,
											   nData	   := _nData,
											   pData	   := _pData,
											   pDoc		   := ValueJson,
											   nDoc		   := SIZEOF(ValueJson),
											   hrErrorCode => hr);

// Attempt to find Member
jsonProp := JsonFileMachineConfig.FindMemberPath(JsonDoc, _SymbolName);
IF JsonProp <> 0 THEN
	JsonFileMachineConfig.SetJson(JsonProp, ValueJson);
ELSE
	JsonFileMachineConfig.AddJsonMember(JsonDoc, _SymbolName, ValueJson);
END_IF

// Save the update to file
FileSave := TRUE;
SeqSave	 := 10;
JsonProp := 0;
END_METHOD

METHOD PRIVATE LoadFileSequence
VAR_INST
	dirPath	 : T_MaxString;
	tryAgain : BOOL;
END_VAR

VAR
	msg : STRING;
END_VAR
CASE SeqLoad OF
	0:										// Attempt to Load File -> Command started in LoadFile()
	10:										// Load File Done
		IF NOT FileRead AND FileLoadOK THEN // File Found
			JsonDoc := JsonFileMachineConfig.GetDocumentRoot();
			SeqLoad := 0;
		END_IF

		IF (NOT FileRead AND NOT FileLoadOK) OR TonTimeout.Q THEN // File not Found
			tryAgain := FALSE;
			FileRead := FALSE;
			SeqLoad	 := 20;
		END_IF

	20:								  (*File Not Found - Create Directory if not exists*) ;
		CreateDir(bExecute := FALSE); //Prepare for rising edge in next step
		IF NOT tryAgain THEN
			dirPath := StringHelper.GetPath(_Path);
		ELSE
			dirPath := StringHelper.GetPath(dirPath);
		END_IF

		SeqLoad := 30;

	30:
		CreateDir(sNetId	:= '',
				  sPathName := dirPath,
				  ePath		:= PATH_GENERIC,
				  bExecute	:= TRUE);

		IF NOT CreateDir.bBusy THEN
			IF NOT CreateDir.bError THEN
				IF NOT tryAgain THEN
					SeqLoad := 40;
				ELSE
					tryAgain := FALSE;
					SeqLoad	 := 20;
				END_IF
			ELSE
				IF (CreateDir.nErrId = 1827) OR (CreateDir.nErrId = 1807) THEN
					//0x723 Folder is already existing or invalid sPathName or ePath parameter.
					msg := CONCAT(_Path, ' File not found, but folder is existing. File will be created');
					Trace.LogMessage(Name, msg);
					SeqLoad := 40;
				ELSIF CreateDir.nErrId = 1804 THEN
					//0x70C Folder not found.
					msg := CONCAT('Folder is not found: ', dirPath);
					msg := CONCAT(msg, ' Reducing Path and trying again.');
					Trace.LogMessage(Name, msg);
					tryagain := TRUE;

					// SeqLoad	 := 20; TwinCat Bug - Ticket BTS-168764 Germany
					SeqLoad := 40;
				ELSE
					msg := CONCAT('Create Directory Error: ', UDINT_TO_STRING(CreateDir.nErrId));
					Trace.LogMessage(Name, msg);
					SeqLoad := 999;
				END_IF
			END_IF
		END_IF

	40: // File not found -> Create file
		JsonDoc	 := JsonFileMachineConfig.NewDocument();
		FileSave := TRUE;
		SeqLoad	 := 50;

	50: // New Document Saved
		IF NOT FileSave AND FileSaveOk THEN
			_Error	:= FALSE;
			SeqLoad := 0;
		END_IF
END_CASE
END_METHOD

METHOD PRIVATE SaveFileSequence
CASE SeqSave OF
	0:	// Attempt to save File -> Command started in UpdateXYZ()
	10: // New Document Saved
		IF NOT FileSave AND FileSaveOk THEN
			SeqSave := 0;
		END_IF
END_CASE
END_METHOD

METHOD Reset
_Error		  := FALSE;
_ErrorId	  := 0;
SeqSave		  := 0;
SeqLoad		  := 0;
TonTimeout.IN := FALSE;
END_METHOD

{attribute 'monitoring' := 'call'}
PROPERTY Busy : BOOL
GET
Busy := SeqSave <> 0 OR SeqLoad <> 0;
END_GET
END_PROPERTY

{attribute 'monitoring' := 'call'}
PROPERTY Error : BOOL
GET
Error := _Error;
END_GET
END_PROPERTY

{attribute 'monitoring' := 'call'}
PROPERTY ErrorId : UDINT
GET
ErrorID := _ErrorID;
END_GET
END_PROPERTY

END_FUNCTION_BLOCK

// Utilities/File/StringHelper
{attribute 'no_explicit_call' := 'This FB is a CLASS and must be accessed using methods or properties'}
FUNCTION_BLOCK StringHelper

METHOD PROTECTED GetExtensionOrVarName : T_MaxString
VAR_INPUT
	input : T_MaxString;
END_VAR

VAR
	i		 : INT;
	charArry : ARRAY[0..255] OF STRING(1);
END_VAR
IF NOT ValidInput(input) THEN
	RETURN;
END_IF

charArry := StringToCharArray(input);
//Get Location of final delimiter '.'
FOR i := LEN(input) - 1 TO 0 BY -1 DO //Start at the end and find the last delimiter
	IF charArry[i] = '.' THEN
		GetExtensionOrVarName := RIGHT(input, LEN(input) - 1 - i);
		EXIT;
	END_IF
END_FOR
END_METHOD

METHOD PROTECTED GetFileNameFromPath : T_MaxString
VAR_INPUT
	input : T_MaxString;
END_VAR

VAR
	i			  : INT;
	searchResults : ARRAY[0..99] OF INT;
	tempPath	  : T_MaxString;
END_VAR
IF NOT ValidInput(input) THEN
	RETURN;
END_IF

tempPath := input; //Copy to temp variable for modification
FOR i := 0 TO LEN(input) - 1 DO
	searchResults[i] := FIND(tempPath, '\');
	IF searchResults[i] > 0 THEN
		tempPath := RIGHT(tempPath, LEN(tempPath) - searchResults[i]); //Remove begining up to and including the first delimiter
	ELSE
		EXIT; //No more delimiters remaining
	END_IF
END_FOR

GetFileNameFromPath := tempPath;
END_METHOD

METHOD PROTECTED GetFilePath : T_MaxString
VAR_INPUT
	input : T_MaxString;
END_VAR

VAR
	tempPath	  : T_MaxString;
	i			  : INT;
	searchResults : ARRAY[0..99] OF INT;
	location	  : INT;
END_VAR
IF NOT ValidInput(input) THEN
	RETURN;
END_IF

tempPath := input;								 //Copy to temp variable for modification
tempPath := LEFT(tempPath, (LEN(tempPath) - 1)); //Remove Last Character, on first pass this has no effect, but on subsequents passes this will remove the ending \

//Reduce String by removing each delimiter and counting number of characters removed to find last '\'
FOR i := 0 TO LEN(input) - 1 DO
	searchResults[i] := FIND(tempPath, '\');
	IF searchResults[i] > 0 THEN
		tempPath := RIGHT(tempPath, LEN(tempPath) - searchResults[i]); //Remove begining up to and including the first delimiter
	ELSE
		EXIT; //No more delimiters remaining
	END_IF
END_FOR

//Sum length of string to last delimiter
FOR i := 0 TO LEN(input) - 1 DO
	IF searchResults[i] > 0 THEN
		location := location + searchResults[i]; //Location of last delimiter
	ELSE
		EXIT;
	END_IF
END_FOR

GetFilePath := LEFT(input, location);
END_METHOD

METHOD GetName : T_MaxString
VAR_INPUT
	FullPath : T_MaxString;
END_VAR
IF NOT ValidInput(FullPath) THEN
	RETURN;
END_IF

//Find the First \ or . to determine if this is a File Path or Symbol Path
IF FIND(FullPath, '\') > 0 THEN
	GetName := GetFileNameFromPath(FullPath);
ELSE //symbolPath
	GetName := GetExtensionOrVarName(FullPath);
END_IF
END_METHOD

METHOD GetPath : T_MaxString
VAR_INPUT
	FullPath : T_MaxString;
END_VAR

VAR
	tempPath : T_MaxString;
END_VAR
IF NOT ValidInput(FullPath) THEN
	RETURN;
END_IF

//Find the First \ or . to determine if this is a File Path or Symbol Path
IF FIND(FullPath, '\') > 0 THEN
	GetPath := GetFilePath(FullPath);
ELSE //symbolPath
	GetPath := GetSymbolPath(FullPath);
END_IF
END_METHOD

METHOD PROTECTED GetSymbolPath : T_MaxString
VAR_INPUT
	input : T_MaxString;
END_VAR

VAR
	i		 : INT;
	charArry : ARRAY[0..255] OF STRING(1);
	tempPath : T_MaxString;
END_VAR
IF NOT ValidInput(input) THEN
	RETURN;
END_IF

charArry := StringToCharArray(input);
tempPath := input;					  //Copy to temp variable for modification
FOR i := LEN(input) - 1 TO 0 BY -1 DO //Start at the end and find the last delimiter
	IF charArry[i] = '.' THEN
		tempPath := LEFT(tempPath, i);
		EXIT;
	END_IF
END_FOR

GetSymbolPath := tempPath;
END_METHOD

METHOD PROTECTED RemoveFirstChar : T_MaxString
VAR_INPUT
	input : T_MaxString;
END_VAR
RemoveFirstChar := DELETE(input, 1, 1);
END_METHOD

METHOD PROTECTED RemoveLastChar : T_MaxString
VAR_INPUT
	input : T_MaxString;
END_VAR
RemoveLastChar := DELETE(input, 1, len(input));
END_METHOD

METHOD PROTECTED StringToCharArray : ARRAY[0..255] OF STRING(1)
VAR_INPUT
	input : T_MaxString;
END_VAR

VAR
	i		 : INT;
	end		 : INT;
	tempPath : T_MaxString;
END_VAR
IF NOT ValidInput(input) THEN
	RETURN;
END_IF

tempPath := input;
//Convert String to CharArray
FOR i := 0 TO LEN(input) - 1 DO
	StringToCharArray[i] := Left(tempPath, 1); //Return the first/next character
	tempPath			 := RemoveFirstChar(tempPath);
END_FOR
END_METHOD

METHOD PROTECTED ValidInput : BOOL
VAR_INPUT
	input : T_MaxString;
END_VAR
IF LEN(input) > 0 THEN
	ValidInput := TRUE;
ELSE
	ValidInput := FALSE;
END_IF
END_METHOD

END_FUNCTION_BLOCK

// Utilities/Flash/SyncedSquareWaves
FUNCTION_BLOCK SyncedSquareWaves EXTENDS CyclicComponent IMPLEMENTS I_Initializable
VAR
	_Initialized  : BOOL;
	PLC_CycleTime : UDINT;
	CycleTime_ms  : LREAL;

	//
	{attribute 'hide'}
	_Wave_500Hz : BOOL;
	{attribute 'hide'}
	_Wave_100Hz : BOOL;
	{attribute 'hide'}
	_Wave_50Hz : BOOL;
	{attribute 'hide'}
	_Wave_5Hz : BOOL;
	{attribute 'hide'}
	_Wave_2Hz : BOOL;
	{attribute 'hide'}
	_Wave_1Hz : BOOL;
	{attribute 'hide'}
	_Wave_0_5Hz : BOOL;
END_VAR

METHOD Initialize
//PLC Scan Info
PLC_CycleTime := TwinCAT_SystemInfoVarList._TaskInfo[GETCURTASKINDEXEX()].CycleTime;
CycleTime_ms  := TO_LREAL(PLC_CycleTime) / 10000.0;

//
_Wave_500Hz	 := TRUE;
_Wave_100Hz	 := TRUE;
_Wave_50Hz	 := TRUE;
_Wave_5Hz	 := TRUE;
_Wave_2Hz	 := TRUE;
_Wave_1Hz	 := TRUE;
_Wave_0_5Hz	 := TRUE;
_Initialized := TRUE;
END_METHOD

{attribute 'monitoring' := 'call'}
PROPERTY Initialized : BOOL
GET
Initialized := _Initialized;
END_GET
SET
_Initialized := Initialized;
END_SET
END_PROPERTY

//! @summary This method serves as the entry point for all underlying FB logic
METHOD PUBLIC CyclicLogic
VAR
	Counter		   : LREAL;
	CountsRequired : LREAL;
	CycleCount	   : UDINT;
END_VAR
IF NOT _Initialized THEN
	Initialize();
	RETURN;
END_IF

CycleCount := TwinCAT_SystemInfoVarList._TaskInfo[GETCURTASKINDEXEX()].CycleCount;
IF (CycleTime_ms <= 1) AND (FRAC(1 / CycleTime_ms) = 0) THEN
	CountsRequired := 1 / CycleTime_ms;
	Counter		   := LMOD(CycleCount, CountsRequired);
	IF (Counter + 1) = CountsRequired THEN
		_Wave_500Hz := NOT _Wave_500Hz;
	END_IF
END_IF

IF (CycleTime_ms <= 5) AND (FRAC(5 / CycleTime_ms) = 0) THEN
	CountsRequired := 5 / CycleTime_ms;
	Counter		   := LMOD(CycleCount, CountsRequired);
	IF (Counter + 1) = CountsRequired THEN
		_Wave_100Hz := NOT _Wave_100Hz;
	END_IF
END_IF

IF (CycleTime_ms <= 10) AND (FRAC(10 / CycleTime_ms) = 0) THEN
	CountsRequired := 10 / CycleTime_ms;
	Counter		   := LMOD(CycleCount, CountsRequired);
	IF (Counter + 1) = CountsRequired THEN
		_Wave_50Hz := NOT _Wave_50Hz;
	END_IF
END_IF

IF (CycleTime_ms <= 100) AND (FRAC(100 / CycleTime_ms) = 0) THEN
	CountsRequired := 100 / CycleTime_ms;
	Counter		   := LMOD(CycleCount, CountsRequired);
	IF (Counter + 1) = CountsRequired THEN
		_Wave_5Hz := NOT _Wave_5Hz;
	END_IF
END_IF

IF (CycleTime_ms <= 250) AND (FRAC(250 / CycleTime_ms) = 0) THEN
	CountsRequired := 250 / CycleTime_ms;
	Counter		   := LMOD(CycleCount, CountsRequired);
	IF (Counter + 1) = CountsRequired THEN
		_Wave_2Hz := NOT _Wave_2Hz;
	END_IF
END_IF

IF (CycleTime_ms <= 500) AND (FRAC(500 / CycleTime_ms) = 0) THEN
	CountsRequired := 500 / CycleTime_ms;
	Counter		   := LMOD(CycleCount, CountsRequired);
	IF (Counter + 1) = CountsRequired THEN
		_Wave_1Hz := NOT _Wave_1Hz;
	END_IF
END_IF

IF (CycleTime_ms <= 1000) AND (FRAC(1000 / CycleTime_ms) = 0) THEN
	CountsRequired := 1000 / CycleTime_ms;
	Counter		   := LMOD(CycleCount, CountsRequired);
	IF (Counter + 1) = CountsRequired THEN
		_Wave_0_5Hz := NOT _Wave_0_5Hz;
	END_IF
END_IF
END_METHOD

{attribute 'monitoring' := 'call'}
PROPERTY Wave_0_5Hz : BOOL
GET
Wave_0_5Hz := _Wave_0_5Hz;
END_GET
END_PROPERTY

{attribute 'monitoring' := 'call'}
PROPERTY Wave_100Hz : BOOL
GET
Wave_100Hz := _Wave_100Hz;
END_GET
END_PROPERTY

{attribute 'monitoring' := 'call'}
PROPERTY Wave_1Hz : BOOL
GET
Wave_1Hz := _Wave_1Hz;
END_GET
END_PROPERTY

{attribute 'monitoring' := 'call'}
PROPERTY Wave_2Hz : BOOL
GET
Wave_2Hz := _Wave_2Hz;
END_GET
END_PROPERTY

{attribute 'monitoring' := 'call'}
PROPERTY Wave_500Hz : BOOL
GET
Wave_500Hz := _Wave_500Hz;
END_GET
END_PROPERTY

{attribute 'monitoring' := 'call'}
PROPERTY Wave_50Hz : BOOL
GET
Wave_50Hz := _Wave_50Hz;
END_GET
END_PROPERTY

{attribute 'monitoring' := 'call'}
PROPERTY Wave_5Hz : BOOL
GET
Wave_5Hz := _Wave_5Hz;
END_GET
END_PROPERTY

END_FUNCTION_BLOCK

// Utilities/Functions/CompareLREAL
FUNCTION CompareLREAL : BOOL
VAR_INPUT
	Var1	: LREAL;
	Var2	: LREAL;
	Epsilon : LREAL := 1E-6;
END_VAR

CompareLREAL := ABS(Var1 - Var2) < Epsilon;

END_FUNCTION

// Utilities/Functions/CompareModulo
FUNCTION CompareModulo : BOOL
VAR_INPUT
	Var1	: LREAL;
	Var2	: LREAL;
	Modulo	: LREAL := 360.0;
	Epsilon : LREAL := 1E-6;
END_VAR

CompareModulo := (ABS(MODABS(Var1, Modulo) - MODABS(Var2, Modulo)) < Epsilon) OR (ABS(MODABS(Var1, Modulo) - MODABS(Var2, Modulo)) > (Modulo - Epsilon));

END_FUNCTION

// Utilities/Functions/PercentToAnalog
FUNCTION PercentToAnalog : INT
VAR_INPUT
	TargetValue : DINT; // 0-100%
END_VAR

PercentToAnalog := TO_INT(32767 * TargetValue / 100);

END_FUNCTION

// Utilities/Timing/Stopwatch
FUNCTION_BLOCK Stopwatch
VAR
	StartTime			: T_DCTIME64;
	EndTime				: T_DCTIME64;
	PreviousLapEndTime	: T_DCTIME64;
	PreviousElapsedTime : LREAL;
	_Running			: BOOL;
END_VAR

VAR CONSTANT
	OneNanosecond : LREAL := 1.0E-9;
END_VAR

{attribute 'monitoring' := 'call'}
PROPERTY Elapsed : LREAL
GET
IF _Running THEN
	Elapsed := TO_LREAL(F_GetCurDcTickTime64() - StartTime) * OneNanosecond;
ELSE
	Elapsed := PreviousElapsedTime;
END_IF
END_GET
END_PROPERTY

METHOD Lap : LREAL;
VAR
	LapEndTime	: T_DCTIME64;
	LapDuration : LREAL;
END_VAR
IF _Running THEN
	LapEndTime		   := F_GetActualDcTime64();
	LapDuration		   := TO_LREAL(LapEndTime - PreviousLapEndTime) * OneNanosecond;
	PreviousLapEndTime := LapEndTime;
	Lap				   := LapDuration;
END_IF
END_METHOD

{attribute 'monitoring' := 'call'}
PROPERTY Running : BOOL
GET
Running := _Running;
END_GET
END_PROPERTY

METHOD Start
StartTime			:= F_GetActualDcTime64();
PreviousLapEndTime	:= StartTime;
_Running			:= TRUE;
PreviousElapsedTime := 0.0;
PreviousElapsedTime := 0;
END_METHOD

METHOD Stop : LREAL
IF _Running THEN
	EndTime				:= F_GetActualDcTime64();
	_Running			:= FALSE;
	PreviousElapsedTime := TO_LREAL(EndTime - StartTime) * OneNanosecond;
	Stop				:= PreviousElapsedTime;
ELSE
	Stop := 0.0;
END_IF
END_METHOD

END_FUNCTION_BLOCK
